(* CODESYS project FU_sMidBIBO.xml

Project tree, tasks and I/O mapping:
  function FU_sMidBIBO [ST]
*)

// FU_sMidBIBO
//This functions extracts a part of a string
// +-----------+----------+----------+-----------------------------------------------------------------------------------------------------------------------+
// |**Version**|**Author**| **Date** |**Changes**                                                                                                            |
// +-----------+----------+----------+-----------------------------------------------------------------------------------------------------------------------+
// | 1         | NSN      | 05-02-19 | Creation                                                                                                              |
// +-----------+----------+----------+-----------------------------------------------------------------------------------------------------------------------+
FUNCTION FU_sMidBIBO : BOOL
VAR_IN_OUT
	sOut		:STRING(1);			//Output String
	sStr		:STRING(1);		//Input String	
END_VAR
VAR_INPUT
	wLen		:WORD;				//Amount to copy
	wPos		:WORD;				//Position to copy from
	wOutSize	:WORD;				//Output String Size
END_VAR
VAR
	InAdd		:POINTER TO BYTE;	//Address of input string
	StrAdd		:POINTER TO BYTE;	//Address of output string
END_VAR

InAdd				:=		ADR(sStr);
StrAdd				:=		ADR(sOut);
IF wPos > 0 THEN
	wPos			:=		wPos - 1;
END_IF
IF wLen > 0 THEN
	WHILE wPos > 0 DO
		wPos		:=		wPos - 1;
		IF InAdd^ = 0 THEN
			RETURN;
		END_IF
		InAdd		:=		InAdd + 1;
	END_WHILE
	WHILE wLen > 0 DO
		wLen		:=		wLen - 1;
		IF InAdd^ = 0 OR wOutSize = 0 THEN
			StrAdd^	:=		0;
			RETURN;
		END_IF
		StrAdd^		:=		InAdd^;
		InAdd		:=		InAdd + 1;
		StrAdd		:=		StrAdd + 1;
		wOutSize	:=		wOutSize - 1;
	END_WHILE
	StrAdd^			:=		0;
END_IF

END_FUNCTION
